// ---- VISUs/Keyboard/Numpad_Original.TcVIS
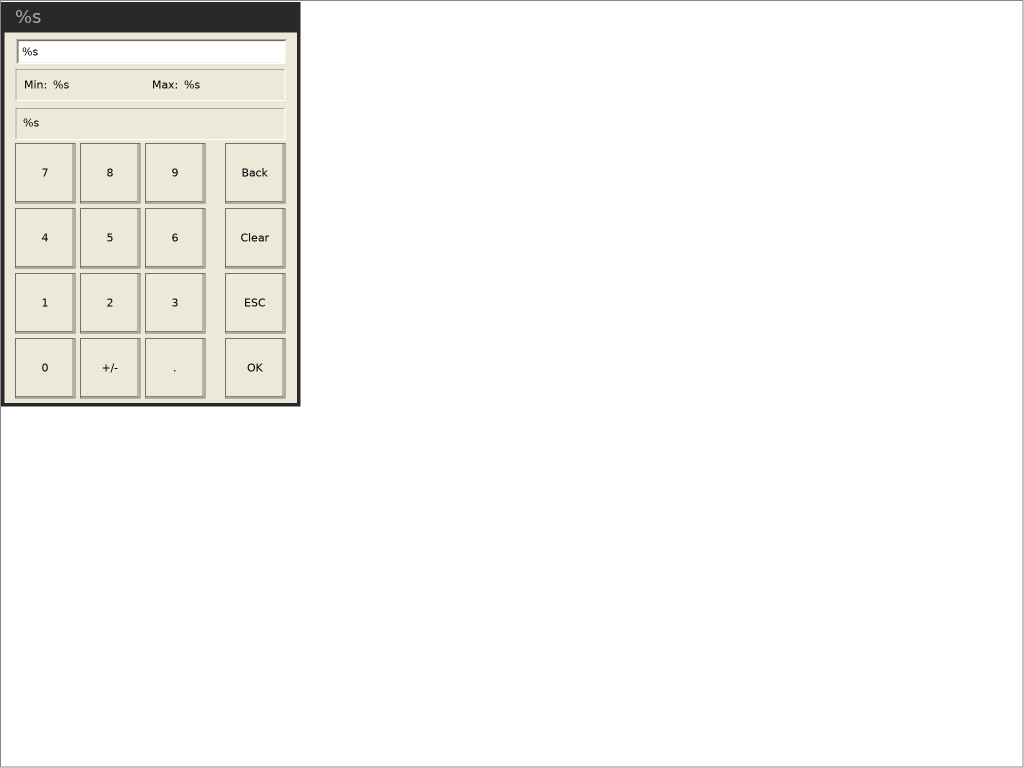
VISUALIZATION Numpad_Original  // 1024x768
VAR_INPUT
	stVariableValue : STRING;
	stMin : STRING;
	stMax : STRING;
	wstTitle : WSTRING;
	flags : DWORD;
END_VAR
VAR
	bInit : BOOL;
	stMessage : STRING;
	stOutputValue : STRING;
	iCaretPosition	: INT;
	iSelectionStart	: INT;
	iSelectionEnd	: INT;
	xAllSelected	: BOOL;
END_VAR
    Rectangle (3,31 294x39)
    Polyline (17,63) (17,39) (286,39)
    Polyline (18,63) (285,63) (285,40)
    Polyline (18,62) (18,40) (285,40)
    Textfield (19,42 265x20), "%s", text variable: stOutputValue
        p905179711: iCaretPosition
        p3815007873: iSelectionStart
        p1425650380: iSelectionEnd
        p3479897389: xAllSelected
    Rectangle (3,138 295x67)
    Rectangle (3,205 295x65)
    Rectangle (3,270 295x65)
    Rectangle (3,335 295x68)
    Button (225,338 60x60), "OK"
        OnMouseDown: CloseDialog Dialog=Numpad, Result=OK, NumpadKeypad=True, NumpadKeypadSet=True
    Button (225,273 60x60), "ESC"
        OnMouseDown: CloseDialog Dialog=Numpad, Result=Cancel, NumpadKeypad=True, NumpadKeypadSet=True
    Button (225,208 60x60), "Clear"
        OnMouseDown: execute {
            stVariableValue := '';
            stOutputValue := '';
            flags := flags AND NOT 16#0008;
            flags := flags AND NOT 16#0010;
            iCaretPosition	:= 1;
            iSelectionStart	:= 1;
            iSelectionEnd	:= 1;
        }
    Button (225,143 60x60), "Back"
        OnMouseDown: execute { VisuDlg_ProcessBack(stOutputValue, stVariableValue, iCaretPosition, iSelectionStart, iSelectionEnd, bInit); }
    Button (145,338 60x60), "."
        OnMouseDown: execute { VisuDlg_ProcessChar(stOutputValue, stVariableValue, iCaretPosition, iSelectionStart, iSelectionEnd, (flags AND VisuElems.Visu_InputFlags.Password) = 1, '.'); }
    Button (80,338 60x60), "+/-"
        OnMouseDown: execute { VisuDlg_ProcessChangeSign(stOutputValue, stVariableValue, iCaretPosition, iSelectionStart, iSelectionEnd, (flags AND VisuElems.Visu_InputFlags.Password) = 1); }
    Button (15,338 60x60), "0"
        OnMouseDown: execute { VisuDlg_ProcessChar(stOutputValue, stVariableValue, iCaretPosition, iSelectionStart, iSelectionEnd, (flags AND VisuElems.Visu_InputFlags.Password) = 1, '0'); }
    Button (15,273 60x60), "1"
        OnMouseDown: execute { VisuDlg_ProcessChar(stOutputValue, stVariableValue, iCaretPosition, iSelectionStart, iSelectionEnd, (flags AND VisuElems.Visu_InputFlags.Password) = 1, '1'); }
    Button (80,273 60x60), "2"
        OnMouseDown: execute { VisuDlg_ProcessChar(stOutputValue, stVariableValue, iCaretPosition, iSelectionStart, iSelectionEnd, (flags AND VisuElems.Visu_InputFlags.Password) = 1, '2'); }
    Button (145,273 60x60), "3"
        OnMouseDown: execute { VisuDlg_ProcessChar(stOutputValue, stVariableValue, iCaretPosition, iSelectionStart, iSelectionEnd, (flags AND VisuElems.Visu_InputFlags.Password) = 1, '3'); }
    Button (15,208 60x60), "4"
        OnMouseDown: execute { VisuDlg_ProcessChar(stOutputValue, stVariableValue, iCaretPosition, iSelectionStart, iSelectionEnd, (flags AND VisuElems.Visu_InputFlags.Password) = 1, '4'); }
    Button (80,208 60x60), "5"
        OnMouseDown: execute { VisuDlg_ProcessChar(stOutputValue, stVariableValue, iCaretPosition, iSelectionStart, iSelectionEnd, (flags AND VisuElems.Visu_InputFlags.Password) = 1, '5'); }
    Button (145,208 60x60), "6"
        OnMouseDown: execute { VisuDlg_ProcessChar(stOutputValue, stVariableValue, iCaretPosition, iSelectionStart, iSelectionEnd, (flags AND VisuElems.Visu_InputFlags.Password) = 1, '6'); }
    Button (15,143 60x60), "7"
        OnMouseDown: execute { VisuDlg_ProcessChar(stOutputValue, stVariableValue, iCaretPosition, iSelectionStart, iSelectionEnd, (flags AND VisuElems.Visu_InputFlags.Password) = 1, '7'); }
    Button (80,143 60x60), "8"
        OnMouseDown: execute { VisuDlg_ProcessChar(stOutputValue, stVariableValue, iCaretPosition, iSelectionStart, iSelectionEnd, (flags AND VisuElems.Visu_InputFlags.Password) = 1, '8'); }
    Button (145,143 60x60), "9"
        OnMouseDown: execute { VisuDlg_ProcessChar(stOutputValue, stVariableValue, iCaretPosition, iSelectionStart, iSelectionEnd, (flags AND VisuElems.Visu_InputFlags.Password) = 1, '9'); }
    Rectangle (3,69 294x69)
    Rectangle (50,75 95x20), "%s", text variable: stMin, invisible if: LEN(stMin) = 0
        p55702900: SEL(((UDINT_TO_DINT(flags AND 16#0008))=16#0008),16#FF000000,16#FFFF0000)
    Rectangle (181,75 95x20), "%s", text variable: stMax, invisible if: LEN(stMax) = 0
        p55702900: SEL(((UDINT_TO_DINT(flags AND 16#0010))=16#0010),16#FF000000,16#FFFF0000)
    Rectangle (149,75 31x20), "Max:", invisible if: LEN(stMax) = 0
        p55702900: SEL(((UDINT_TO_DINT(flags AND 16#0010))=16#0010),16#FF000000,16#FFFF0000)
    Rectangle (296,403 3x3)
    Rectangle (297,2 3x404)
    Rectangle (1,3 3x403)
    Rectangle (1,2 298x30), invisible if: VisuElems.g_VisualizationStyle.GetDINT('Dialog-UseHeaderColor', 0, 0) = 0
    Rectangle (12,7 280x20), "%s", text variable: wstTitle
    Rectangle (1,403 299x3)
    Polyline (16,138) (16,108) (284,108)
    Polyline (16,99) (16,69) (284,69)
    Polyline (17,139) (285,139) (285,108)
    Polyline (17,100) (285,100) (285,69)
    Rectangle (20,113 95x20), "%s", text variable: stMessage
    Rectangle (21,75 31x20), "Min:", invisible if: LEN(stMin) = 0
        p55702900: SEL(((UDINT_TO_DINT(flags AND 16#0008))=16#0008),16#FF000000,16#FFFF0000)
END_VISUALIZATION

// ---- VISUs/vMain.TcVIS
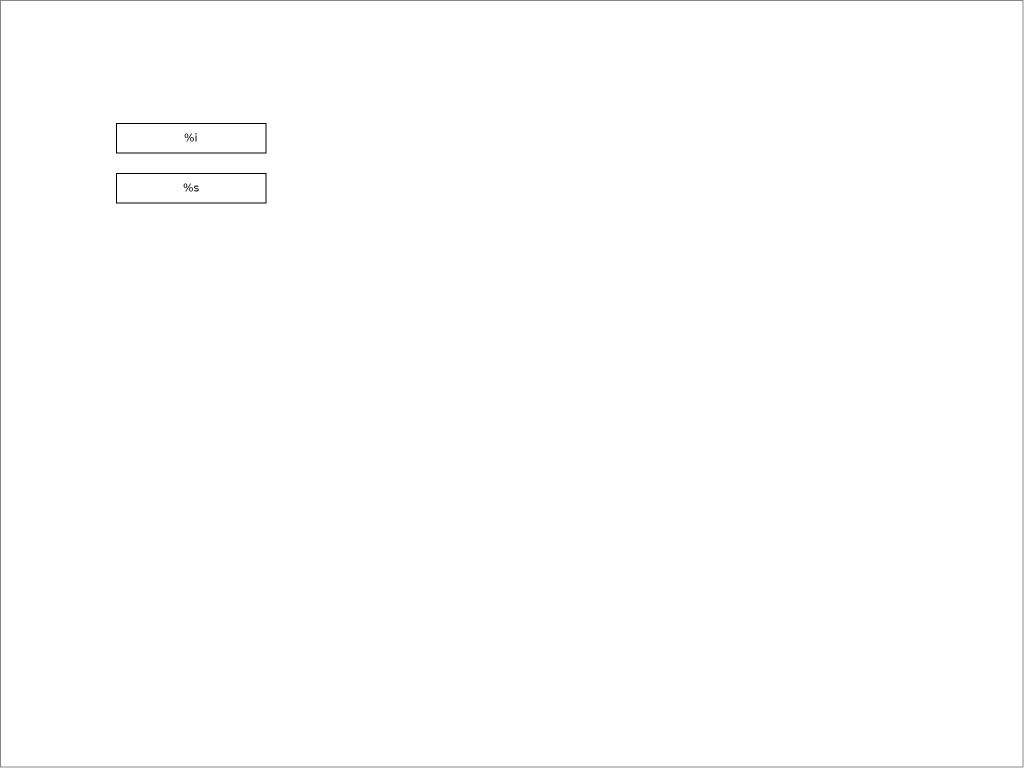
VISUALIZATION vMain  // 1024x768
    Rectangle (116,123 150x30), "%i", text variable: MAIN.nTest
        OnMouseDown: execute { gsPadTitle := 'Numpad nTest'; }
        OnMouseDown: write the text variable via Numpad
    Rectangle (116,173 150x30), "%s", text variable: MAIN.sTest
        OnMouseDown: execute { gsPadTitle := 'Keypad sTest'; }
        OnMouseDown: write the text variable via Keypad
END_VISUALIZATION
